{attribute 'qualified_only'}
{attribute 'strict'}
TYPE
    eCustomizedDialogAnswer :
    (
        NoAnswer := 0,
        Option1 := 10,
        Option2 := 20,
        Option3 := 30,
        Option4 := 40
    );
END_TYPE

(* stored: Version 1.1.0.1
   DUT eCustomizedDialogAnswer: Id {d8ccb112-c774-059b-10fc-addce03e14ac} *)
